// TIA Portal V17 export
// export: Created 2025-06-26T06:49:13.5079766Z, ExportSetting WithDefaults, DisplayName Totally Integrated Automation Portal, DisplayVersion V17 Update 8, DisplayName TIA Portal Openness, DisplayVersion V17 Update 8, DisplayName TIA Portal Version Control Interface, DisplayVersion V17, DisplayName STEP 7 Professional, DisplayVersion V17 Update 8, DisplayName STEP 7 Safety, DisplayVersion V17 Update 6, DisplayName WinCC Advanced, DisplayVersion V17 Update 8
FUNCTION_BLOCK "StartStopControl"   // FB30, FBD
{ S7_Optimized_Access := 'TRUE' }
VERSION : 0.1
// stored: AutoNumber true, IsIECCheckEnabled false, IsRetainMemResEnabled false, MemoryReserve 0, SetENOAutomatically false, UDAEnableTagReadback false
   VAR_OUTPUT
      Run : Bool;   // 1 = run, 0 = stop
   END_VAR
   VAR
      StartRequestHMI { ExternalAccessible := 'False'; ExternalVisible := 'False'; ExternalWritable := 'False'; S7_SetPoint := 'True'} : R_TRIG;
      StartRequestApplication { ExternalAccessible := 'False'; ExternalVisible := 'False'; ExternalWritable := 'False'; S7_SetPoint := 'True'} : R_TRIG;
      StopRequestHMI { ExternalAccessible := 'False'; ExternalVisible := 'False'; ExternalWritable := 'False'; S7_SetPoint := 'True'} : R_TRIG;
      StopRequestApplication { ExternalAccessible := 'False'; ExternalVisible := 'False'; ExternalWritable := 'False'; S7_SetPoint := 'True'} : R_TRIG;
      EmergencyStopWaitTime { S7_SetPoint := 'True'} : TOF_TIME;
      StopRequestCriticalAlarm { S7_SetPoint := 'True'} : Bool;
   END_VAR
   VAR_TEMP
      StopRequestRegulatorFault : Bool;
   END_VAR
BEGIN

REGION Network 1: Start request signals
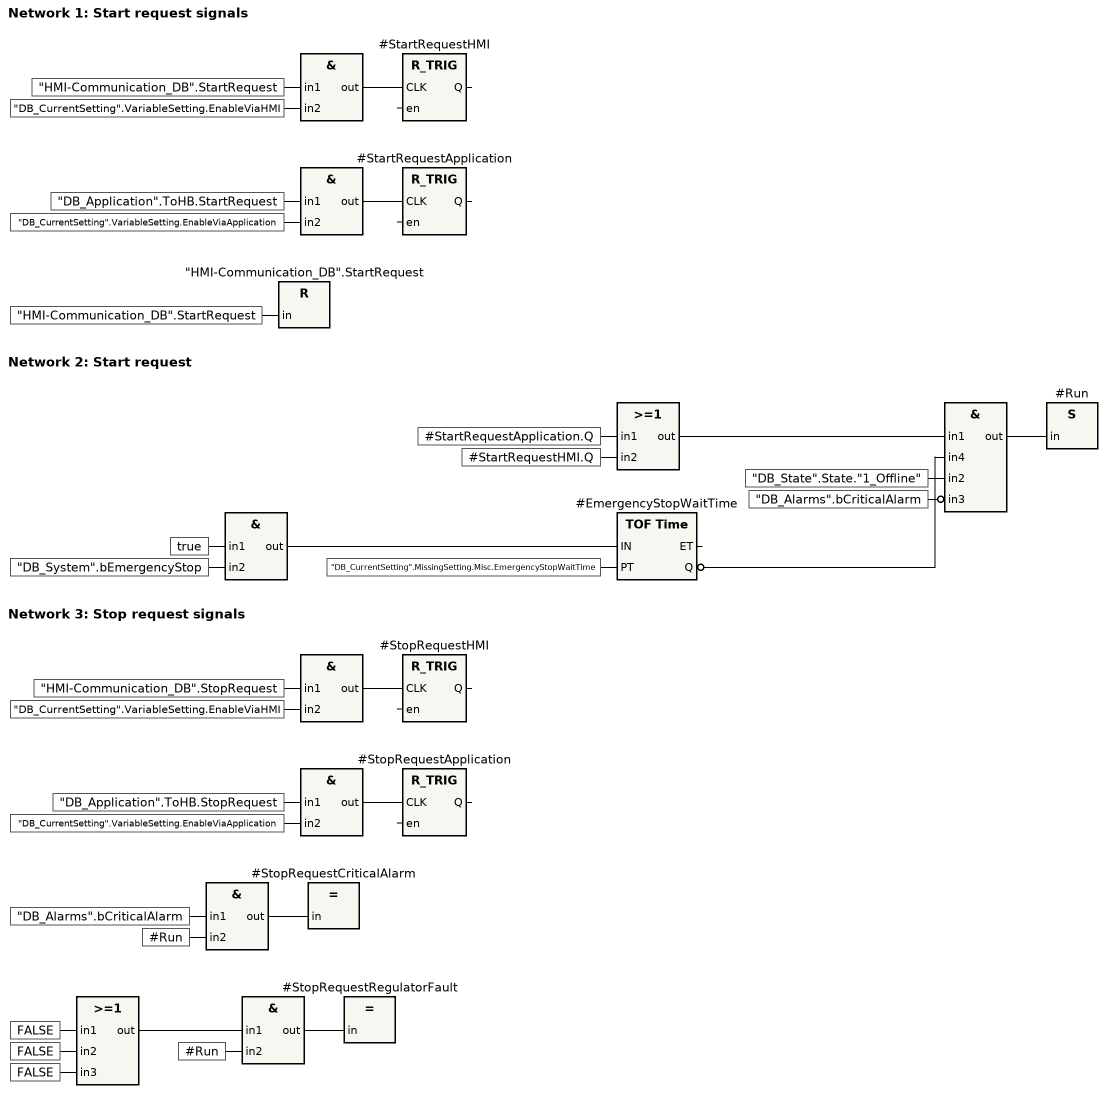
   #StartRequestHMI(CLK := "HMI-Communication_DB".StartRequest AND "DB_CurrentSetting".VariableSetting.EnableViaHMI);   // R_TRIG
   #StartRequestApplication(CLK := "DB_Application".ToHB.StartRequest AND "DB_CurrentSetting".VariableSetting.EnableViaApplication);   // R_TRIG
   IF "HMI-Communication_DB".StartRequest THEN "HMI-Communication_DB".StartRequest := FALSE; END_IF;
END_REGION

REGION Network 2: Start request
   // Start conditions:
   // 1. Start request from one of the control sources
   // 2. State 1 
   // 3. No critical alarms active
   // 4. E-stop lockout timer has expired
   // Also reset alarms
   #EmergencyStopWaitTime(IN := true AND "DB_System".bEmergencyStop,   // TOF
                          PT := "DB_CurrentSetting".MissingSetting.Misc.EmergencyStopWaitTime);
   IF (#StartRequestApplication.Q OR #StartRequestHMI.Q) AND NOT #EmergencyStopWaitTime.Q AND "DB_State".State."1_Offline" AND NOT "DB_Alarms".bCriticalAlarm THEN
       #Run := TRUE;
   END_IF;
END_REGION

REGION Network 3: Stop request signals
   // ##FIX decide what to do about regulator faults.
   #StopRequestHMI(CLK := "HMI-Communication_DB".StopRequest AND "DB_CurrentSetting".VariableSetting.EnableViaHMI);   // R_TRIG
   #StopRequestApplication(CLK := "DB_Application".ToHB.StopRequest AND "DB_CurrentSetting".VariableSetting.EnableViaApplication);   // R_TRIG
   #StopRequestCriticalAlarm := "DB_Alarms".bCriticalAlarm AND #Run;
   #StopRequestRegulatorFault := (FALSE OR FALSE OR FALSE) AND #Run;
END_REGION

REGION Network 4: Stop request
   // Stop condition is one of:
   // 1. Stop request from one of the control sources (HMI or App PLC)
   // 2. Forced into State 7 Stop (and the machine should follow)
   // 3. Critical Alarm
   // 4. Emergency Stop. (This is also technically a critical alarm but alarms can be disabled)
   // 5. Regulator fault
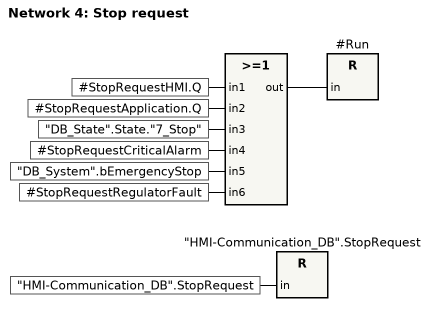
   IF #StopRequestHMI.Q OR #StopRequestApplication.Q OR "DB_State".State."7_Stop" OR #StopRequestCriticalAlarm OR "DB_System".bEmergencyStop OR #StopRequestRegulatorFault THEN
       #Run := FALSE;
   END_IF;
   IF "HMI-Communication_DB".StopRequest THEN "HMI-Communication_DB".StopRequest := FALSE; END_IF;
END_REGION
END_FUNCTION_BLOCK
